Staubli VAL3: onF5Event.pgx

program onF5Event()
  local num l_nSize
begin
  // look if the bButton is enable
  if bButton[4]
    //
    // select/ unselect the items
    //
    call prog:selectItem(nIndex)
    call prog:getSizeItem(l_nSize)
    // go down
    if nIndex<l_nSize-1
      nSelected=nId+1
    endIf
    call buildList()
  endIf
end
